Staubli VAL3: TrajJointItem.pjx

--- TrajJointItem.pjx ---
Parameters version=s7.2.1 stackSize=5000 millimeterUnit=true
Data file=TrajJointItem.dtx
Type name=TrajectoryItem path=Disk://kernel/template/TrajectoryItem/TrajectoryItem.pjx

--- TrajJointItem.dtx ---
public jointRx jJoint
public TrajectoryItem tSuper
  [0]
    num distance
    num moveType
    num nTime
    num nStop
    num nTcpAction
    string comment
    bool toStop
    mdesc nom_speed = {tmax=300, rmax=9999, leave=30, reach=30}
    InstrItem iInstr[3]
      [0]
        string sType
        string sData
      [1]
        string sType
        string sData
      [2]
        string sType
        string sData
    num nMoveId
